FUNCTION_BLOCK FB_ControllerType_2 IMPLEMENTS InterfaceFuture
VAR_INPUT
END_VAR
VAR_OUTPUT
END_VAR
VAR
	_own_parameter: UINT;
	process_timer: TON;
	blink_timer: TON;
	_result :HRESULT;
	_counter :UINT;
END_VAR
VAR_IN_OUT
	own_input: BOOL;
	own_output: BOOL;
END_VAR

{warning 'add property implementation'}
PROPERTY active_futures : UINT
GET
END_GET
END_PROPERTY

PROPERTY counter : UINT
GET
counter := _counter;
END_GET
END_PROPERTY

METHOD execute : BOOL
VAR_INPUT
END_VAR
VAR_INST
	input_memory :BOOL;
END_VAR
own_output := TRUE;
IF own_input AND NOT input_memory THEN
	_counter := counter + 1;
END_IF
input_memory := own_input;
IF _counter > _own_parameter THEN
	execute := TRUE;
END_IF
END_METHOD

METHOD init : BOOL
VAR_INPUT
END_VAR
own_output := FALSE;
process_timer(IN := FALSE);
blink_timer(IN := FALSE);
_counter := 0;
init := TRUE;
END_METHOD

PROPERTY own_parameter : UINT
GET
own_parameter := _own_parameter;
END_GET
SET
_own_parameter := own_parameter;
END_SET
END_PROPERTY

{warning 'add method implementation '}
METHOD quit : BOOL
THIS^.init();
quit := TRUE;
END_METHOD

{warning 'add property implementation'}
PROPERTY result : HRESULT
GET
result := _result;
END_GET
END_PROPERTY

END_FUNCTION_BLOCK

(* stored: Version 1.1.0.1, ProductVersion 3.1.4024.12
   POU FB_ControllerType_2: Id {fcedd839-491a-4b82-962e-a6b212add423}, SpecialFunc None
   Property active_futures: Id {faf0be87-65d0-4052-a2bd-7d503c7aeb21}
   Get Get: Id {f75d49fc-753d-4d3e-960d-ee7e63a88e67}
   Property counter: Id {d21e7cd7-0ef0-4123-a4e3-71fe9855b00a}
   Get Get: Id {a2a1935b-4339-4663-9b2a-10527d776baa}
   Method execute: Id {06ca504b-2230-462e-b402-b0513637b891}
   Method init: Id {0506fa37-b033-4ecf-a1b9-39ffd68590c2}
   Property own_parameter: Id {44c22855-b665-42b9-9698-003553798c6b}
   Get Get: Id {a4ce69b5-d711-41f1-b7ea-5a7f1940c7a1}
   Set Set: Id {20314786-f00f-435f-bd37-c1bd1124cdd5}
   Method quit: Id {77d78392-ba97-4c0d-a7ef-71aa64534b7c}
   Property result: Id {16e63a23-0f02-402f-9998-37a3e09307d6}
   Get Get: Id {10902b3b-ec3f-43fc-b121-362377561d1c} *)
